# EPICS substitutions: ipimbIocApp/Db/autosave_ipimbIoc.substitutions
#
# ipimbIoc substitutions file
#

# Generate iocAdmin autosave request
file autosave_iocAdmin.template
{
	{
		# Hack till msi supports empty substitutions
		_FOOBAR_=_FOOBAR_
	}
}
